// TIA Portal V20 export
TYPE "typeEm0Standard"
// stored: Access Published, Namespace Unit1
   STRUCT
      commands { ExternalWritable := 'False'} : "Unit1.typeEm0Commands";
      monitoring { ExternalWritable := 'False'} : "Unit1.typeEm0Monitoring";
   END_STRUCT;
END_TYPE
